VAR_GLOBAL
	PLCEtherCatAddress : T_AmsNetId;
END_VAR

(* stored: Version 1.1.0.1, ProductVersion 3.1.4024.10
   GVL GVL: Id {c5a6c953-0a19-4476-a183-82196d385398} *)
